{attribute addProperty BoxType "KL6224-0003"}
{attribute addProperty Id "Channel_1Channel_0418AA5000"}
{attribute addProperty CRC "3328131575"}
{attribute addProperty SizeInBites "0"}
{attribute addProperty SizeInBytes "0"}
TYPE KL_C65F41F7 :
STRUCT
	{attribute addProperty Name "Channel_1"}
	Channel_1 : Channel_0418AA50;
END_STRUCT
END_TYPE

(* stored: Version 1.2.0.0, ProductVersion 3.1.4024.9
   DUT KL_C65F41F7: Id {b48c103a-0b5b-472d-8eab-b2914085068a} *)
